// TIA Portal V19 export
FUNCTION "Input Toggle" : Void   // FC2, LAD
{ S7_Optimized_Access := 'TRUE' }
// stored: SetENOAutomatically false
   VAR_IN_OUT
      Toggle_Input : Bool;
   END_VAR
BEGIN

REGION Network 1
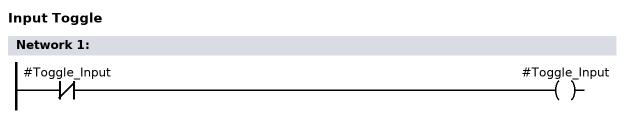
   RUNG wire#powerrail
      I_Contact( #Toggle_Input )
      Coil( #Toggle_Input )
   END_RUNG
   // the same network as SCL:
   #Toggle_Input := NOT #Toggle_Input;
END_REGION
END_FUNCTION
